{attribute addProperty BoxType "AX5106-0000-0010-0010"}
{attribute addProperty Id "AT_xAT %I*AT_x_029F01154860MDTAT %Q*MDT_47A878CF4860WcStateAT %I*WcState_F855686C1620InfoDataAT %I*InfoData_AEB17F4D152190"}
{attribute addProperty CRC "237890021"}
{attribute addProperty SizeInBites "264"}
{attribute addProperty SizeInBytes "33"}
TYPE AX5106_3F57D30F :
STRUCT
	{attribute addProperty Name "AT_x"}
	AT_x : AT_x_029F0115;
	{attribute addProperty Name "MDT"}
	MDT : MDT_47A878CF;
	{attribute addProperty Name "WcState"}
	WcState : WcState_F855686C;
	{attribute addProperty Name "InfoData"}
	InfoData : InfoData_AEB17F4D;
END_STRUCT
END_TYPE

(* stored: Version 1.2.0.0, ProductVersion 3.1.4024.9
   DUT AX5106_3F57D30F: Id {f1badf08-d84e-4a89-99ec-d8402ccd3edc} *)
